(* Logix 5000 project; controller IF2_DEMO Emulate 5570 rev 20.12; software revision 20.04; part 5 of 8 *)
(* tags used below, declared in another part *)
   CIP_String_Creator : STRING;
   CIP_TimeStamp : STRING;
   CIP_TimeStamp_Day : STRING;
   CIP_TimeStamp_Month : STRING;
   CIPActive : BOOL;
   CIPAlarm_Start : BOOL;
   CIPAlarmTrigger : BOOL[32];
   CIPClarity : DINT;
   CIPFilling : BOOL[32];
   CIPTimer : TIMER[4];
   CIPValve0 : ALARM_DIGITAL;
   CIPValve1 : ALARM_DIGITAL;
   CIPValve2 : ALARM_DIGITAL;
   CIPValve3 : ALARM_DIGITAL;
   Delay : TIMER[4];
   DispenserLine : LineData;
   HMISystemClock : DINT[7];
   Menu_GOTO_dx : DINT;
   Menu_GOTO_H : DINT;
   Menu_GOTO_POS : DINT;
   MotorOverheatAlarm : ALARM_ANALOG;
   MotorTemp : DINT;
   Phase_1 : PHASE;
   Phase_2 : PHASE;
   Phase_Timer : TIMER;
   RefillLine : LineData;
   Run_Day : INT;
   Run_Hr : INT;
   Run_Min : INT;
   Run_Sec : INT;
   Run_Timer : TIMER;
   SodaCIPTanks : IPTankLevel;
   TankValue : DINT[4];
   Timer1000ms : TIMER;
   Timer100ms : TIMER;
   Timer10ms : TIMER;
   Timer1ms : TIMER;
   Timer250ms : TIMER;
   Timer500ms : TIMER;
   TimeTrigger : BOOL;
   ValveFlowOn : BOOL;
   WallClock : DINT[7];
   WC : WC[10];

PROGRAM Main   (* main routine MainRoutine *)
VAR
   Agitator : DISCRETE_2STATE := (State0Perm := 1, State1Perm := 1);
   Alarm_RapidMixStopped : ALARM_DIGITAL;
   ApplyDSTBit : DINT := 1;
   Assembly : MotionVars := (Motion := 9.0, MotionFactor := 3.0, MotionMax := 99.0);
   Blending_Discharge_Jam_Tank1 : ALARM_DIGITAL;
   Blending_Discharge_Tank1_Jam_Ack : BOOL := 1;
   Blending_Discharge_Tank1_Jam_Ind : BOOL := 1;
   Blending_Discharge_Tank1_Jam_Timer_Sim : TIMER := (PRE := 500004, ACC := 253104, EN := 1, TT := 1);
   CIP_Clarify_Sensor_Ack : BOOL;
   CIP_Clarify_Sensor_Ind : BOOL;
   CIP_Clarify_Sensor_Timer_Sim : TIMER := (PRE := 1100022, ACC := 653241, EN := 1, TT := 1);
   CIP_Clarity_Sensor : ALARM_DIGITAL;
   CIP_Drain_Valve : ALARM_DIGITAL;
   CIP_Drain_Valve_Ack : BOOL;
   CIP_Drain_Valve_Ind : BOOL;
   CIP_Drain_Valve_Timer_Sim : TIMER := (PRE := 900000, ACC := 53334, EN := 1, TT := 1);
   CIP_Supply_Motor : ALARM_ANALOG;
   CIP_Supply_Motor_Ack : BOOL;
   CIP_Supply_Motor_Ind : BOOL;
   CIP_Supply_Motor_Timer_Sim : TIMER := (PRE := 900001, ACC := 53325, EN := 1, TT := 1);
   CIP_TimeStamp_ONS : BOOL;
   CIPSteps : DINT := 5;
   Complete_Manual_Step_AUTO : TIMER := (PRE := 240000);
   Filler_Valve_3a_Ack : BOOL;
   Filler_Valve_3a_Ind : BOOL;
   Filler_Valve_3a_Timer_Sim : TIMER := (PRE := 301000, ACC := 28908, EN := 1, TT := 1);
   Filler_Valve_6B_Ack : BOOL;
   Filler_Valve_6B_Ind : BOOL;
   Filler_Valve_6B_Timer_Sim : TIMER := (PRE := 400000, ACC := 53031, EN := 1, TT := 1);
   Filling_Valve_3a : ALARM_DIGITAL;
   Filling_Valve_3a_Ack : BOOL;
   Filling_Valve_6b : ALARM_DIGITAL;
   Labeler_Motor : ALARM_ANALOG;
   Labeler_Motor_Ack : BOOL;
   Labeler_Motor_Timer_Sim : TIMER := (PRE := 200019, ACC := 51885, EN := 1, TT := 1);
   Main : MotionVars := (Motion := 30.0, MotionFactor := 1.0, MotionMax := 100.0);
   Maximum : DINT[4] := ([0] := 20000, [1] := 20000, [2] := 20000, [3] := 20000);
   Mixer_Step_6_AUTORESET : TIMER := (PRE := 15000);
   Packaging_Motor : ALARM_ANALOG;
   Packaging_Motor_Ack : BOOL;
   Packaging_Motor_Timer_Sim : TIMER := (PRE := 300222, ACC := 47541, EN := 1, TT := 1);
   Paint : MotionVars := (MotionFactor := 1.0, MotionMax := 199.0);
   repeatCIP : BOOL;
   Restart_CIP_Timer_AUTO : TIMER := (PRE := 150000, ACC := 123517, EN := 1, TT := 1);
   TempCalc : DINT[4] := ([0] := 12500, [1] := 20000, [2] := 1982, [3] := 2000);
   TempCalc2 : DINT[4] := ([0] := 20000, [1] := 20000, [2] := 7982, [3] := 8000);
   test_bit : BOOL := 1;
   Test_Pack : MotionVars := (Motion := 39.0, MotionFactor := 3.0, MotionMax := 49.0);
   Test_Toggle : BOOL;
   TestLatch : BOOL;
   trig : DINT := 20686;
   xUtility : TIMER := (PRE := 500, ACC := 313, EN := 1, TT := 1);
   xUtilityBit : DINT;
END_VAR

ROUTINE Alarms   (* ladder *)
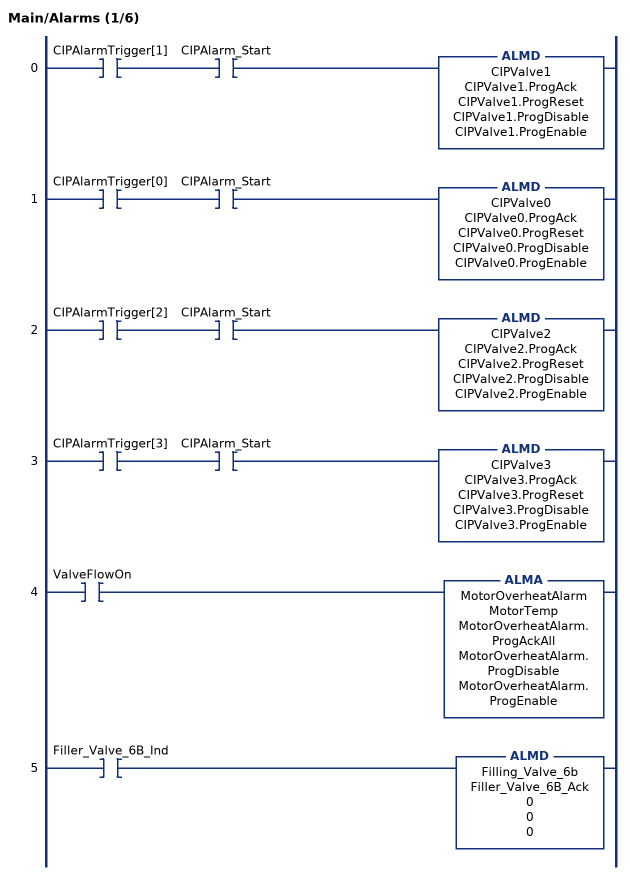
   0: XIC(CIPAlarmTrigger[1])XIC(CIPAlarm_Start)ALMD(CIPValve1,CIPValve1.ProgAck,CIPValve1.ProgReset,CIPValve1.ProgDisable,CIPValve1.ProgEnable);
   1: XIC(CIPAlarmTrigger[0])XIC(CIPAlarm_Start)ALMD(CIPValve0,CIPValve0.ProgAck,CIPValve0.ProgReset,CIPValve0.ProgDisable,CIPValve0.ProgEnable);
   2: XIC(CIPAlarmTrigger[2])XIC(CIPAlarm_Start)ALMD(CIPValve2,CIPValve2.ProgAck,CIPValve2.ProgReset,CIPValve2.ProgDisable,CIPValve2.ProgEnable);
   3: XIC(CIPAlarmTrigger[3])XIC(CIPAlarm_Start)ALMD(CIPValve3,CIPValve3.ProgAck,CIPValve3.ProgReset,CIPValve3.ProgDisable,CIPValve3.ProgEnable);
   4: XIC(ValveFlowOn)ALMA(MotorOverheatAlarm,MotorTemp,MotorOverheatAlarm.ProgAckAll,MotorOverheatAlarm.ProgDisable,MotorOverheatAlarm.ProgEnable);
   5: XIC(Filler_Valve_6B_Ind)ALMD(Filling_Valve_6b,Filler_Valve_6B_Ack,0,0,0);
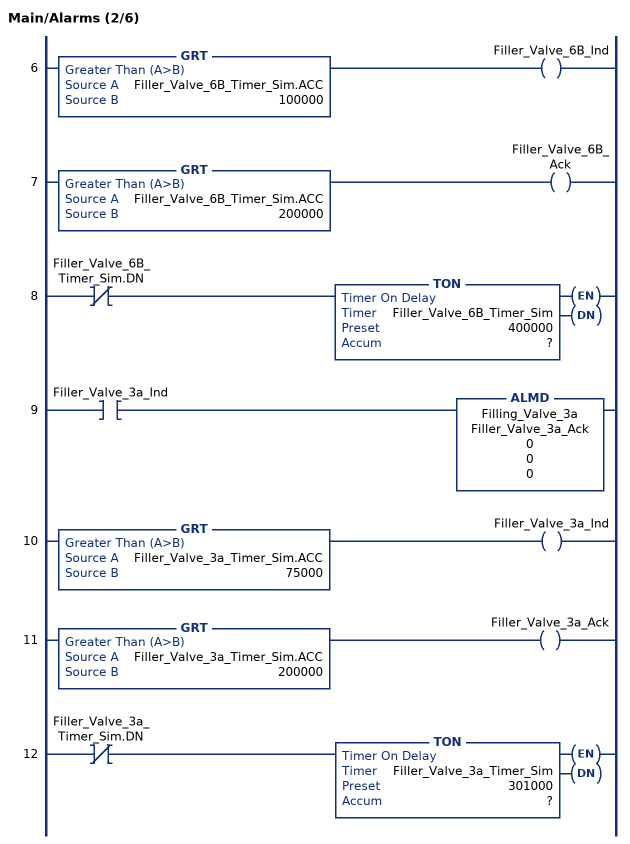
   6: GRT(Filler_Valve_6B_Timer_Sim.ACC,100000)OTE(Filler_Valve_6B_Ind);
   7: GRT(Filler_Valve_6B_Timer_Sim.ACC,200000)OTE(Filler_Valve_6B_Ack);
   8: XIO(Filler_Valve_6B_Timer_Sim.DN)TON(Filler_Valve_6B_Timer_Sim,?,?);
   9: XIC(Filler_Valve_3a_Ind)ALMD(Filling_Valve_3a,Filler_Valve_3a_Ack,0,0,0);
   10: GRT(Filler_Valve_3a_Timer_Sim.ACC,75000)OTE(Filler_Valve_3a_Ind);
   11: GRT(Filler_Valve_3a_Timer_Sim.ACC,200000)OTE(Filler_Valve_3a_Ack);
   12: XIO(Filler_Valve_3a_Timer_Sim.DN)TON(Filler_Valve_3a_Timer_Sim,?,?);
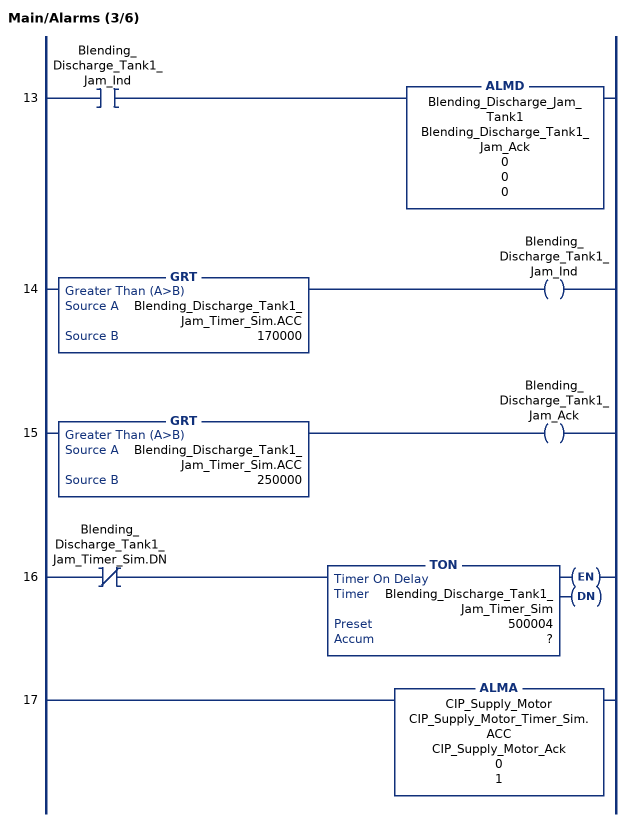
   13: XIC(Blending_Discharge_Tank1_Jam_Ind)ALMD(Blending_Discharge_Jam_Tank1,Blending_Discharge_Tank1_Jam_Ack,0,0,0);
   14: GRT(Blending_Discharge_Tank1_Jam_Timer_Sim.ACC,170000)OTE(Blending_Discharge_Tank1_Jam_Ind);
   15: GRT(Blending_Discharge_Tank1_Jam_Timer_Sim.ACC,250000)OTE(Blending_Discharge_Tank1_Jam_Ack);
   16: XIO(Blending_Discharge_Tank1_Jam_Timer_Sim.DN)TON(Blending_Discharge_Tank1_Jam_Timer_Sim,?,?);
   17: ALMA(CIP_Supply_Motor,CIP_Supply_Motor_Timer_Sim.ACC,CIP_Supply_Motor_Ack,0,1);
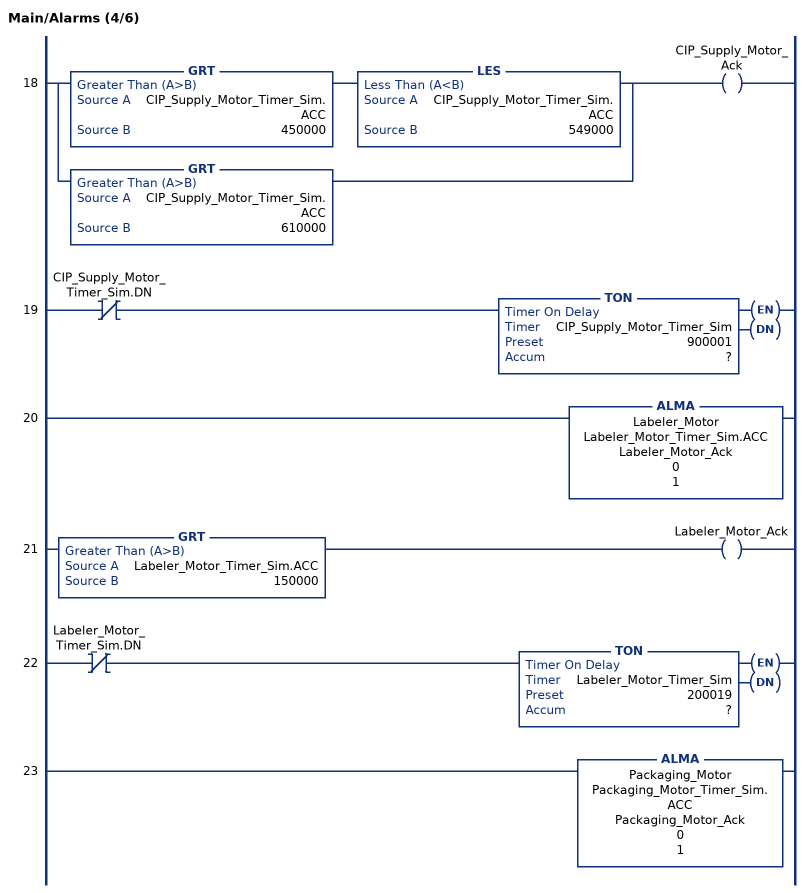
   18: [GRT(CIP_Supply_Motor_Timer_Sim.ACC,450000) LES(CIP_Supply_Motor_Timer_Sim.ACC,549000) ,GRT(CIP_Supply_Motor_Timer_Sim.ACC,610000) ]OTE(CIP_Supply_Motor_Ack);
   19: XIO(CIP_Supply_Motor_Timer_Sim.DN)TON(CIP_Supply_Motor_Timer_Sim,?,?);
   20: ALMA(Labeler_Motor,Labeler_Motor_Timer_Sim.ACC,Labeler_Motor_Ack,0,1);
   21: GRT(Labeler_Motor_Timer_Sim.ACC,150000)OTE(Labeler_Motor_Ack);
   22: XIO(Labeler_Motor_Timer_Sim.DN)TON(Labeler_Motor_Timer_Sim,?,?);
   23: ALMA(Packaging_Motor,Packaging_Motor_Timer_Sim.ACC,Packaging_Motor_Ack,0,1);
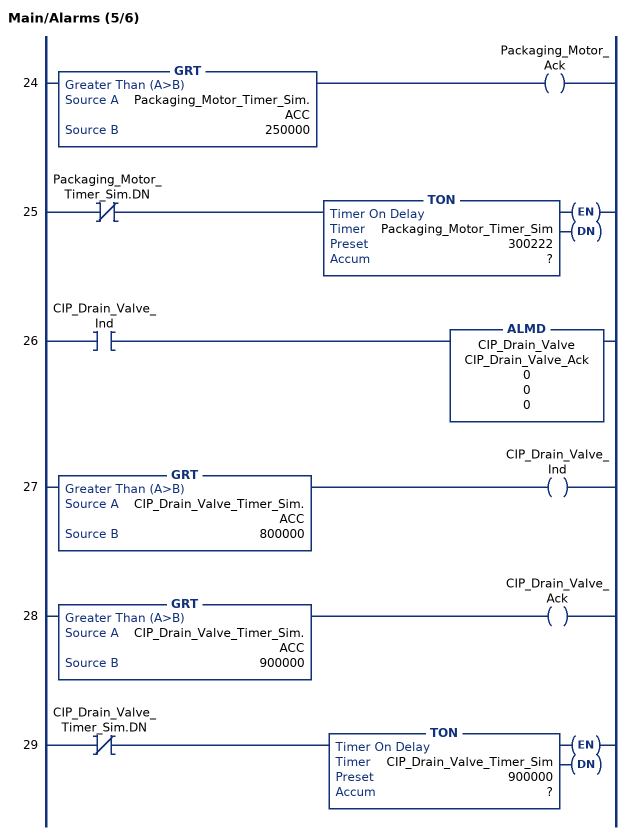
   24: GRT(Packaging_Motor_Timer_Sim.ACC,250000)OTE(Packaging_Motor_Ack);
   25: XIO(Packaging_Motor_Timer_Sim.DN)TON(Packaging_Motor_Timer_Sim,?,?);
   26: XIC(CIP_Drain_Valve_Ind)ALMD(CIP_Drain_Valve,CIP_Drain_Valve_Ack,0,0,0);
   27: GRT(CIP_Drain_Valve_Timer_Sim.ACC,800000)OTE(CIP_Drain_Valve_Ind);
   28: GRT(CIP_Drain_Valve_Timer_Sim.ACC,900000)OTE(CIP_Drain_Valve_Ack);
   29: XIO(CIP_Drain_Valve_Timer_Sim.DN)TON(CIP_Drain_Valve_Timer_Sim,?,?);
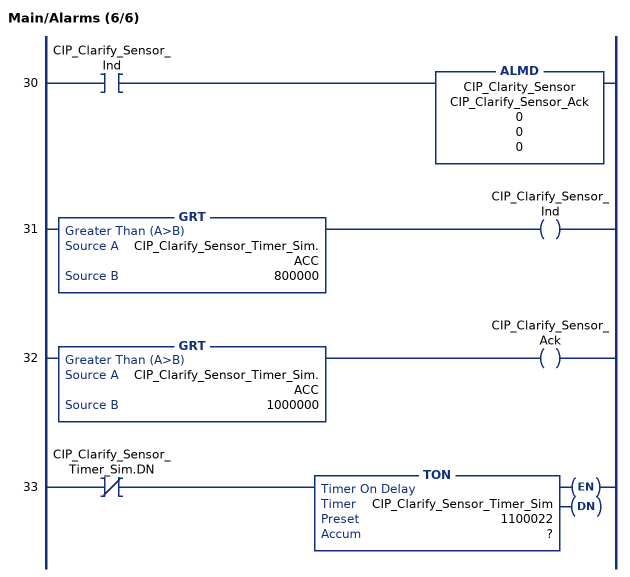
   30: XIC(CIP_Clarify_Sensor_Ind)ALMD(CIP_Clarity_Sensor,CIP_Clarify_Sensor_Ack,0,0,0);
   31: GRT(CIP_Clarify_Sensor_Timer_Sim.ACC,800000)OTE(CIP_Clarify_Sensor_Ind);
   32: GRT(CIP_Clarify_Sensor_Timer_Sim.ACC,1000000)OTE(CIP_Clarify_Sensor_Ack);
   33: XIO(CIP_Clarify_Sensor_Timer_Sim.DN)TON(CIP_Clarify_Sensor_Timer_Sim,?,?);
END_ROUTINE

ROUTINE CIP   (* ladder *)
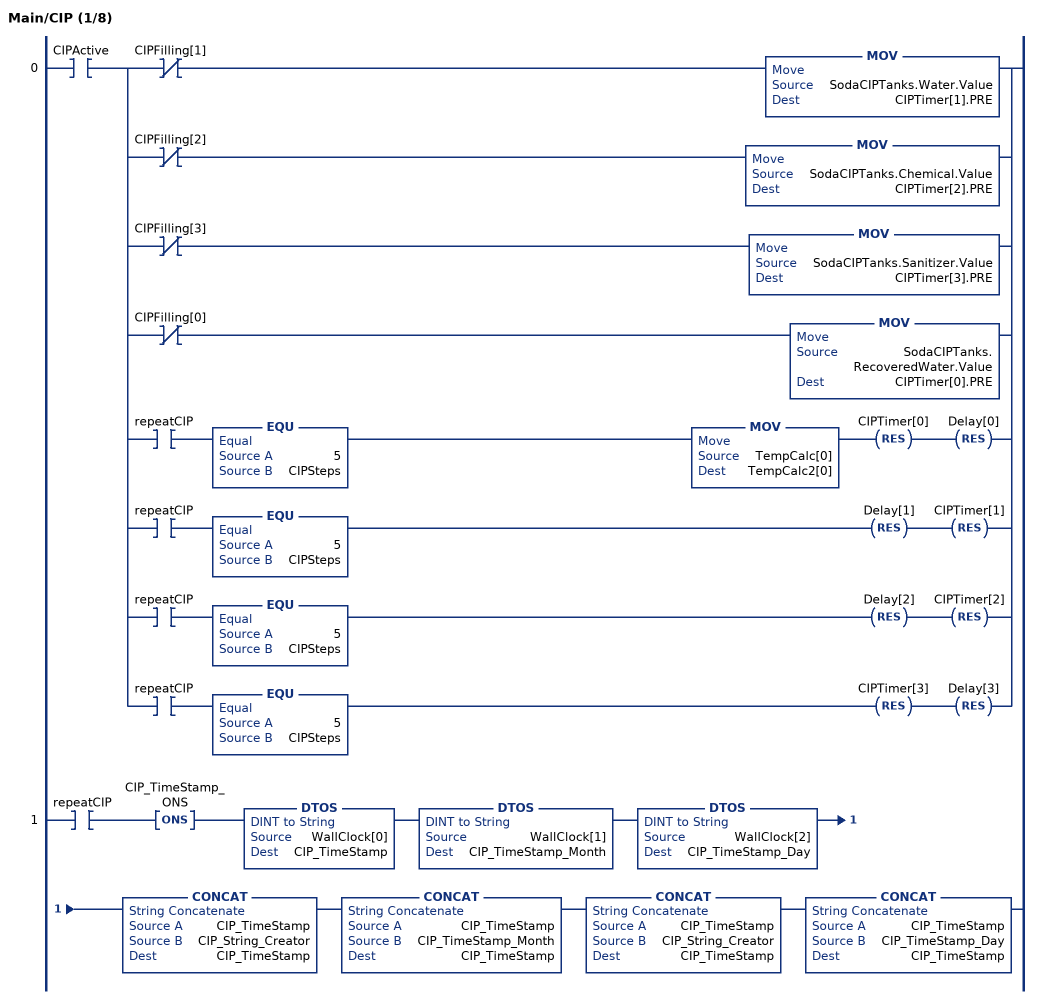
   0: XIC(CIPActive)[XIO(CIPFilling[1]) MOV(SodaCIPTanks.Water.Value,CIPTimer[1].PRE) ,[XIO(CIPFilling[2]) MOV(SodaCIPTanks.Chemical.Value,CIPTimer[2].PRE) ,XIO(CIPFilling[3]) MOV(SodaCIPTanks.Sanitizer.Value,CIPTimer[3].PRE) ,XIO(CIPFilling[0]) MOV(SodaCIPTanks.RecoveredWater.Value,CIPTimer[0].PRE) ,XIC(repeatCIP) EQU(5,CIPSteps) MOV(TempCalc[0],TempCalc2[0]) RES(CIPTimer[0]) RES(Delay[0]) ,XIC(repeatCIP) EQU(5,CIPSteps) RES(Delay[1]) RES(CIPTimer[1]) ,XIC(repeatCIP) EQU(5,CIPSteps) RES(Delay[2]) RES(CIPTimer[2]) ,XIC(repeatCIP) EQU(5,CIPSteps) RES(CIPTimer[3]) RES(Delay[3]) ] ];
   1: XIC(repeatCIP)ONS(CIP_TimeStamp_ONS)DTOS(WallClock[0],CIP_TimeStamp)DTOS(WallClock[1],CIP_TimeStamp_Month)DTOS(WallClock[2],CIP_TimeStamp_Day)CONCAT(CIP_TimeStamp,CIP_String_Creator,CIP_TimeStamp)CONCAT(CIP_TimeStamp,CIP_TimeStamp_Month,CIP_TimeStamp)CONCAT(CIP_TimeStamp,CIP_String_Creator,CIP_TimeStamp)CONCAT(CIP_TimeStamp,CIP_TimeStamp_Day,CIP_TimeStamp);
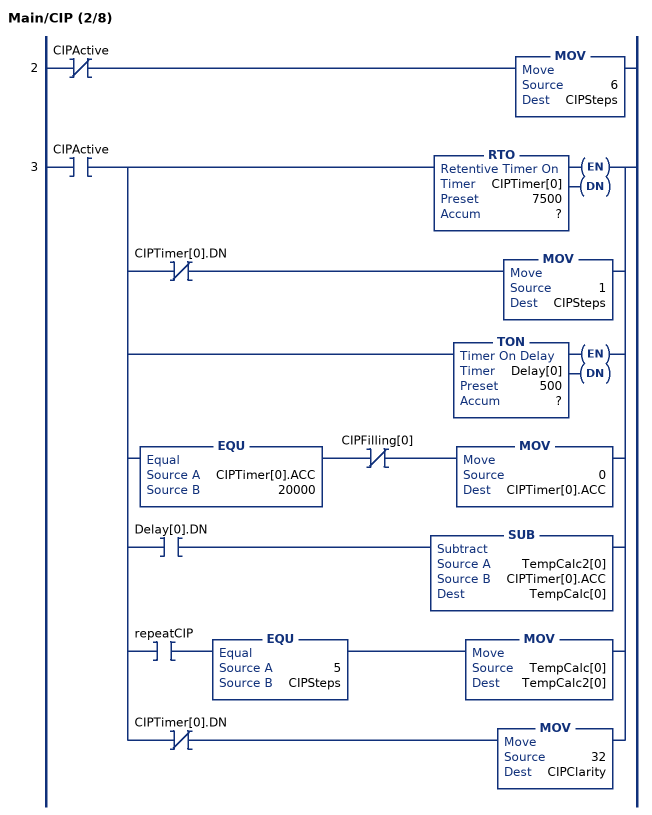
   2: XIO(CIPActive)MOV(6,CIPSteps);
   3: XIC(CIPActive)[RTO(CIPTimer[0],?,?) ,XIO(CIPTimer[0].DN) MOV(1,CIPSteps) ,TON(Delay[0],?,?) ,EQU(CIPTimer[0].ACC,20000) XIO(CIPFilling[0]) MOV(0,CIPTimer[0].ACC) ,XIC(Delay[0].DN) SUB(TempCalc2[0],CIPTimer[0].ACC,TempCalc[0]) ,XIC(repeatCIP) EQU(5,CIPSteps) MOV(TempCalc[0],TempCalc2[0]) ,XIO(CIPTimer[0].DN) MOV(32,CIPClarity) ];
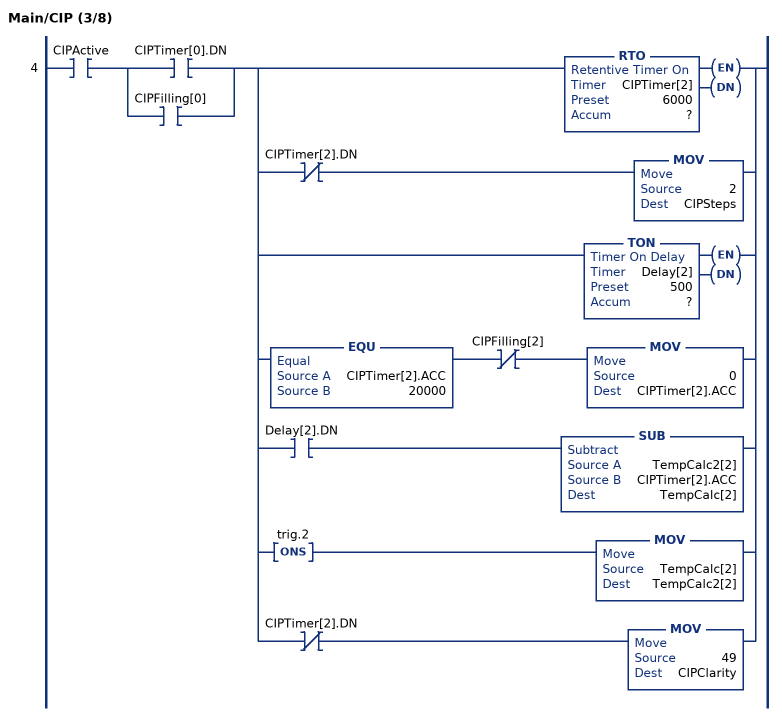
   4: XIC(CIPActive)[XIC(CIPTimer[0].DN) ,XIC(CIPFilling[0]) ][RTO(CIPTimer[2],?,?) ,XIO(CIPTimer[2].DN) MOV(2,CIPSteps) ,TON(Delay[2],?,?) ,EQU(CIPTimer[2].ACC,20000) XIO(CIPFilling[2]) MOV(0,CIPTimer[2].ACC) ,XIC(Delay[2].DN) SUB(TempCalc2[2],CIPTimer[2].ACC,TempCalc[2]) ,ONS(trig.2) MOV(TempCalc[2],TempCalc2[2]) ,XIO(CIPTimer[2].DN) MOV(49,CIPClarity) ];
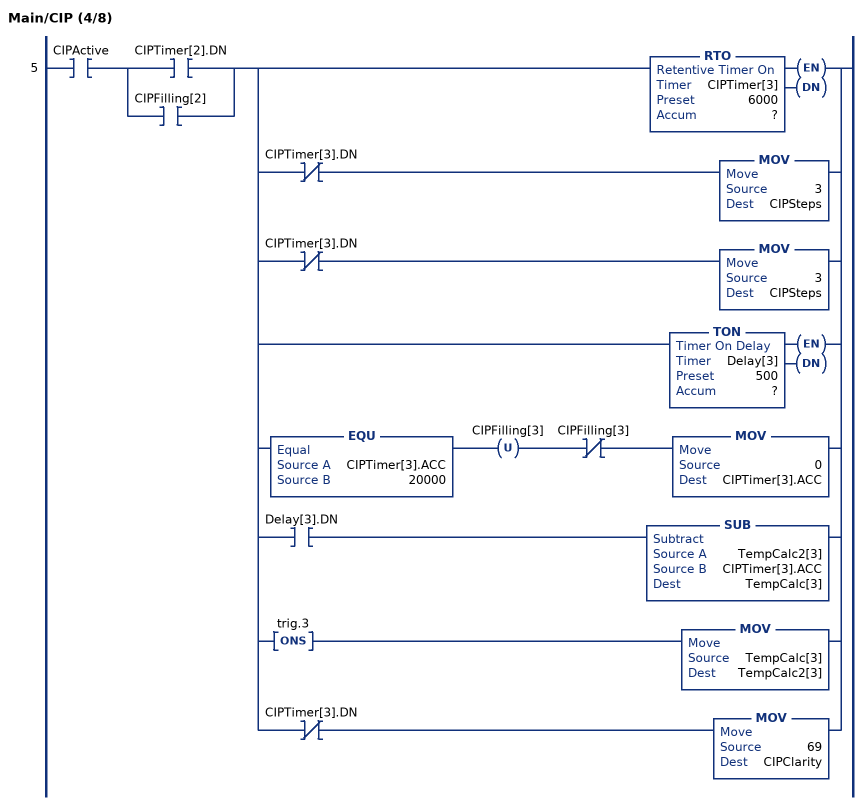
   5: XIC(CIPActive)[XIC(CIPTimer[2].DN) ,XIC(CIPFilling[2]) ][RTO(CIPTimer[3],?,?) ,XIO(CIPTimer[3].DN) MOV(3,CIPSteps) ,XIO(CIPTimer[3].DN) MOV(3,CIPSteps) ,TON(Delay[3],?,?) ,EQU(CIPTimer[3].ACC,20000) OTU(CIPFilling[3]) XIO(CIPFilling[3]) MOV(0,CIPTimer[3].ACC) ,XIC(Delay[3].DN) SUB(TempCalc2[3],CIPTimer[3].ACC,TempCalc[3]) ,ONS(trig.3) MOV(TempCalc[3],TempCalc2[3]) ,XIO(CIPTimer[3].DN) MOV(69,CIPClarity) ];
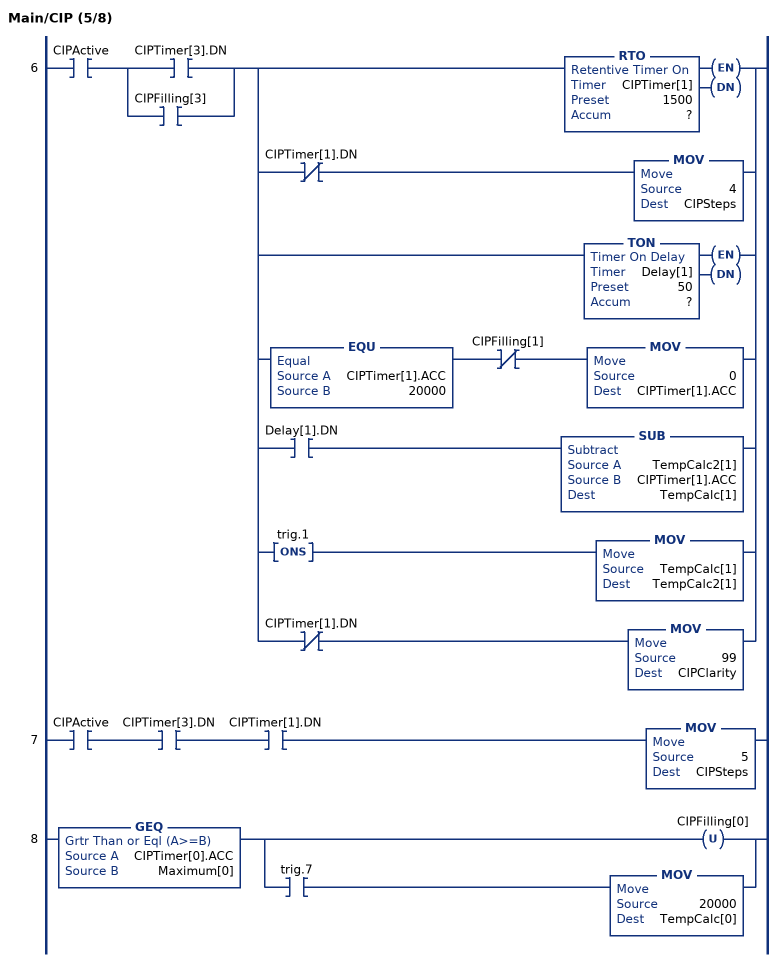
   6: XIC(CIPActive)[XIC(CIPTimer[3].DN) ,XIC(CIPFilling[3]) ][RTO(CIPTimer[1],?,?) ,XIO(CIPTimer[1].DN) MOV(4,CIPSteps) ,TON(Delay[1],?,?) ,EQU(CIPTimer[1].ACC,20000) XIO(CIPFilling[1]) MOV(0,CIPTimer[1].ACC) ,XIC(Delay[1].DN) SUB(TempCalc2[1],CIPTimer[1].ACC,TempCalc[1]) ,ONS(trig.1) MOV(TempCalc[1],TempCalc2[1]) ,XIO(CIPTimer[1].DN) MOV(99,CIPClarity) ];
   7: XIC(CIPActive)XIC(CIPTimer[3].DN)XIC(CIPTimer[1].DN)MOV(5,CIPSteps);
   8: GEQ(CIPTimer[0].ACC,Maximum[0])[OTU(CIPFilling[0]) ,XIC(trig.7) MOV(20000,TempCalc[0]) ];
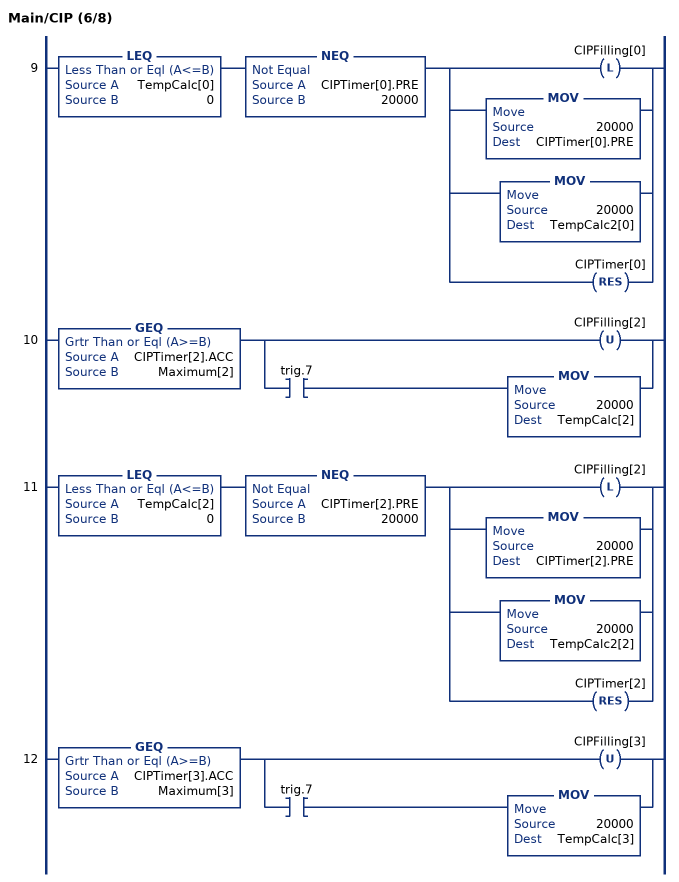
   9: LEQ(TempCalc[0],0)NEQ(CIPTimer[0].PRE,20000)[OTL(CIPFilling[0]) ,MOV(20000,CIPTimer[0].PRE) ,MOV(20000,TempCalc2[0]) ,RES(CIPTimer[0]) ];
   10: GEQ(CIPTimer[2].ACC,Maximum[2])[OTU(CIPFilling[2]) ,XIC(trig.7) MOV(20000,TempCalc[2]) ];
   11: LEQ(TempCalc[2],0)NEQ(CIPTimer[2].PRE,20000)[OTL(CIPFilling[2]) ,MOV(20000,CIPTimer[2].PRE) ,MOV(20000,TempCalc2[2]) ,RES(CIPTimer[2]) ];
   12: GEQ(CIPTimer[3].ACC,Maximum[3])[OTU(CIPFilling[3]) ,XIC(trig.7) MOV(20000,TempCalc[3]) ];
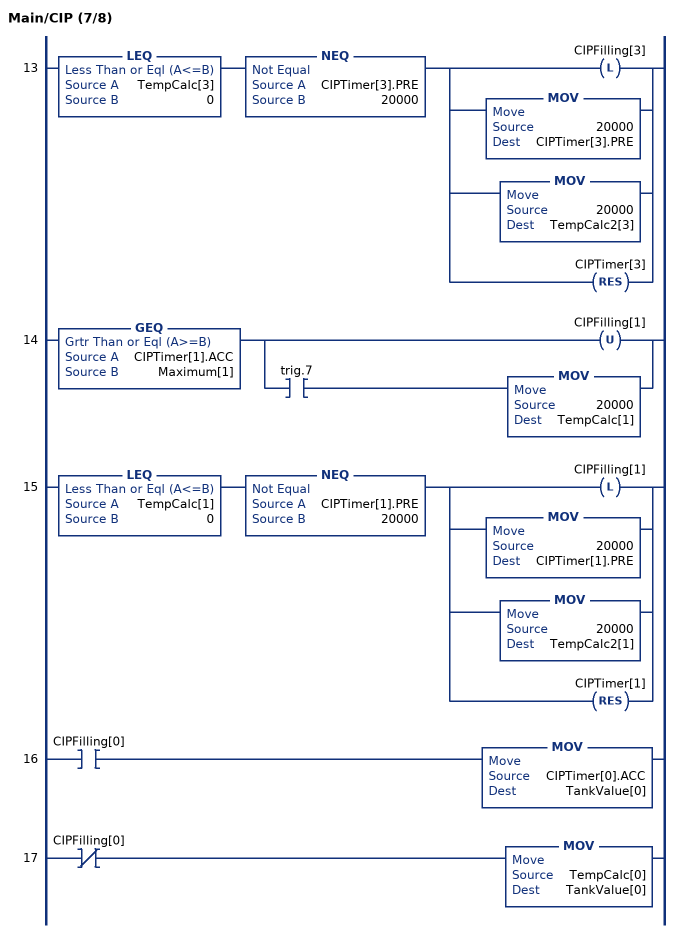
   13: LEQ(TempCalc[3],0)NEQ(CIPTimer[3].PRE,20000)[OTL(CIPFilling[3]) ,MOV(20000,CIPTimer[3].PRE) ,MOV(20000,TempCalc2[3]) ,RES(CIPTimer[3]) ];
   14: GEQ(CIPTimer[1].ACC,Maximum[1])[OTU(CIPFilling[1]) ,XIC(trig.7) MOV(20000,TempCalc[1]) ];
   15: LEQ(TempCalc[1],0)NEQ(CIPTimer[1].PRE,20000)[OTL(CIPFilling[1]) ,MOV(20000,CIPTimer[1].PRE) ,MOV(20000,TempCalc2[1]) ,RES(CIPTimer[1]) ];
   16: XIC(CIPFilling[0])MOV(CIPTimer[0].ACC,TankValue[0]);
   17: XIO(CIPFilling[0])MOV(TempCalc[0],TankValue[0]);
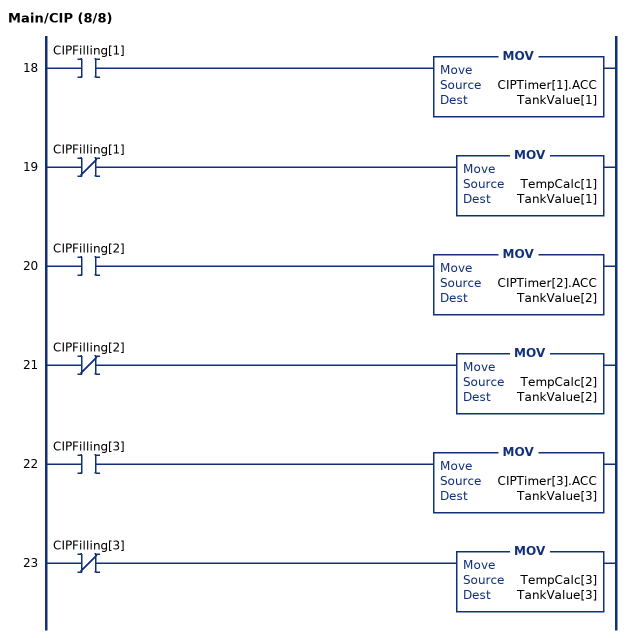
   18: XIC(CIPFilling[1])MOV(CIPTimer[1].ACC,TankValue[1]);
   19: XIO(CIPFilling[1])MOV(TempCalc[1],TankValue[1]);
   20: XIC(CIPFilling[2])MOV(CIPTimer[2].ACC,TankValue[2]);
   21: XIO(CIPFilling[2])MOV(TempCalc[2],TankValue[2]);
   22: XIC(CIPFilling[3])MOV(CIPTimer[3].ACC,TankValue[3]);
   23: XIO(CIPFilling[3])MOV(TempCalc[3],TankValue[3]);
END_ROUTINE

ROUTINE MainRoutine   (* ladder *)
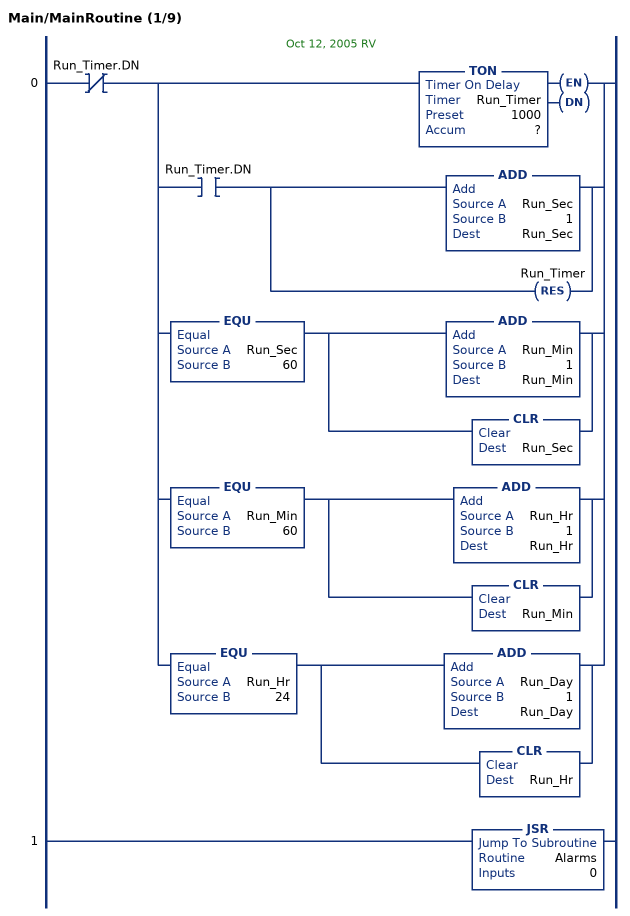
   // Oct 12, 2005 RV
   0: XIO(Run_Timer.DN)[TON(Run_Timer,?,?) ,XIC(Run_Timer.DN) [ADD(Run_Sec,1,Run_Sec) ,RES(Run_Timer) ] ,EQU(Run_Sec,60) [ADD(Run_Min,1,Run_Min) ,CLR(Run_Sec) ] ,EQU(Run_Min,60) [ADD(Run_Hr,1,Run_Hr) ,CLR(Run_Min) ] ,EQU(Run_Hr,24) [ADD(Run_Day,1,Run_Day) ,CLR(Run_Hr) ] ];
   1: JSR(Alarms,0);
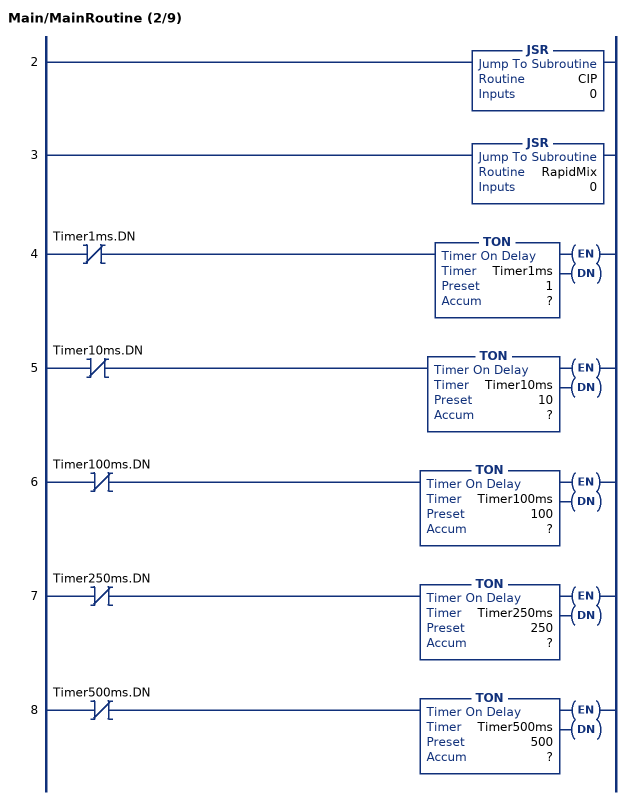
   2: JSR(CIP,0);
   3: JSR(RapidMix,0);
   4: XIO(Timer1ms.DN)TON(Timer1ms,?,?);
   5: XIO(Timer10ms.DN)TON(Timer10ms,?,?);
   6: XIO(Timer100ms.DN)TON(Timer100ms,?,?);
   7: XIO(Timer250ms.DN)TON(Timer250ms,?,?);
   8: XIO(Timer500ms.DN)TON(Timer500ms,?,?);
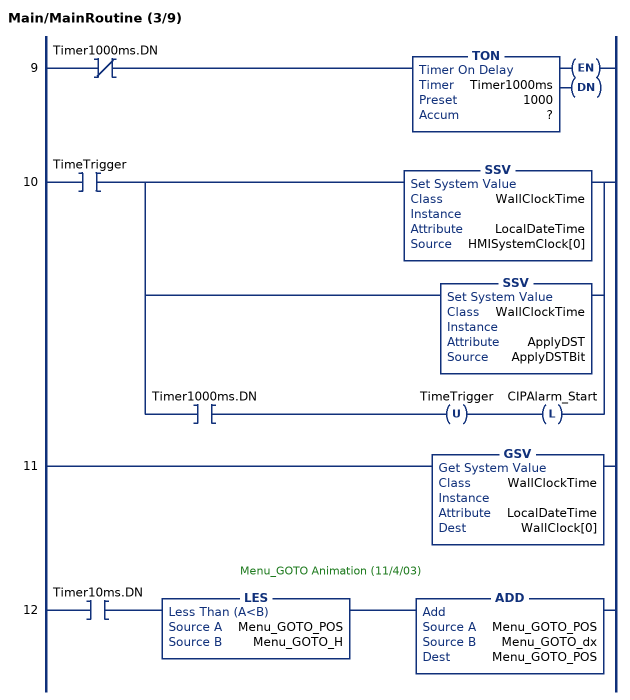
   9: XIO(Timer1000ms.DN)TON(Timer1000ms,?,?);
   10: XIC(TimeTrigger)[SSV(WallClockTime,,LocalDateTime,HMISystemClock[0]) ,SSV(WallClockTime,,ApplyDST,ApplyDSTBit) ,XIC(Timer1000ms.DN) OTU(TimeTrigger) OTL(CIPAlarm_Start) ];
   11: GSV(WallClockTime,,LocalDateTime,WallClock[0]);
   // Menu_GOTO Animation (11/4/03)
   12: XIC(Timer10ms.DN)LES(Menu_GOTO_POS,Menu_GOTO_H)ADD(Menu_GOTO_POS,Menu_GOTO_dx,Menu_GOTO_POS);
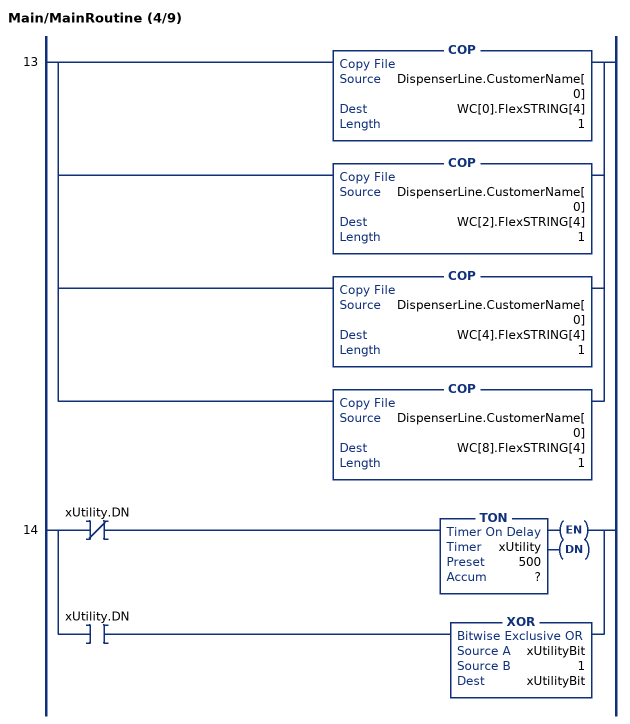
   13: [COP(DispenserLine.CustomerName[0],WC[0].FlexSTRING[4],1) ,COP(DispenserLine.CustomerName[0],WC[2].FlexSTRING[4],1) ,COP(DispenserLine.CustomerName[0],WC[4].FlexSTRING[4],1) ,COP(DispenserLine.CustomerName[0],WC[8].FlexSTRING[4],1) ];
   14: [XIO(xUtility.DN) TON(xUtility,?,?) ,XIC(xUtility.DN) XOR(xUtilityBit,1,xUtilityBit) ];
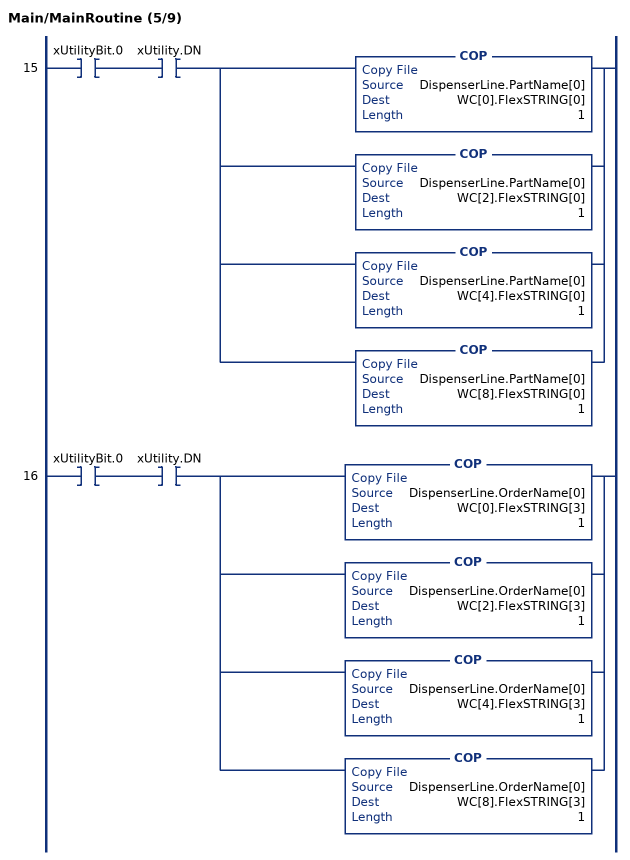
   15: XIC(xUtilityBit.0)XIC(xUtility.DN)[COP(DispenserLine.PartName[0],WC[0].FlexSTRING[0],1) ,COP(DispenserLine.PartName[0],WC[2].FlexSTRING[0],1) ,COP(DispenserLine.PartName[0],WC[4].FlexSTRING[0],1) ,COP(DispenserLine.PartName[0],WC[8].FlexSTRING[0],1) ];
   16: XIC(xUtilityBit.0)XIC(xUtility.DN)[COP(DispenserLine.OrderName[0],WC[0].FlexSTRING[3],1) ,COP(DispenserLine.OrderName[0],WC[2].FlexSTRING[3],1) ,COP(DispenserLine.OrderName[0],WC[4].FlexSTRING[3],1) ,COP(DispenserLine.OrderName[0],WC[8].FlexSTRING[3],1) ];
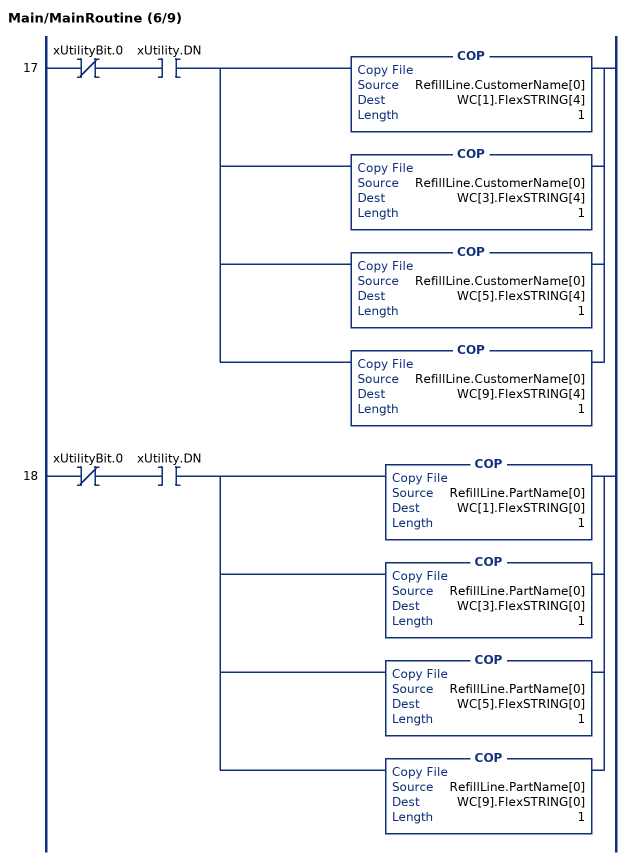
   17: XIO(xUtilityBit.0)XIC(xUtility.DN)[COP(RefillLine.CustomerName[0],WC[1].FlexSTRING[4],1) ,COP(RefillLine.CustomerName[0],WC[3].FlexSTRING[4],1) ,COP(RefillLine.CustomerName[0],WC[5].FlexSTRING[4],1) ,COP(RefillLine.CustomerName[0],WC[9].FlexSTRING[4],1) ];
   18: XIO(xUtilityBit.0)XIC(xUtility.DN)[COP(RefillLine.PartName[0],WC[1].FlexSTRING[0],1) ,COP(RefillLine.PartName[0],WC[3].FlexSTRING[0],1) ,COP(RefillLine.PartName[0],WC[5].FlexSTRING[0],1) ,COP(RefillLine.PartName[0],WC[9].FlexSTRING[0],1) ];
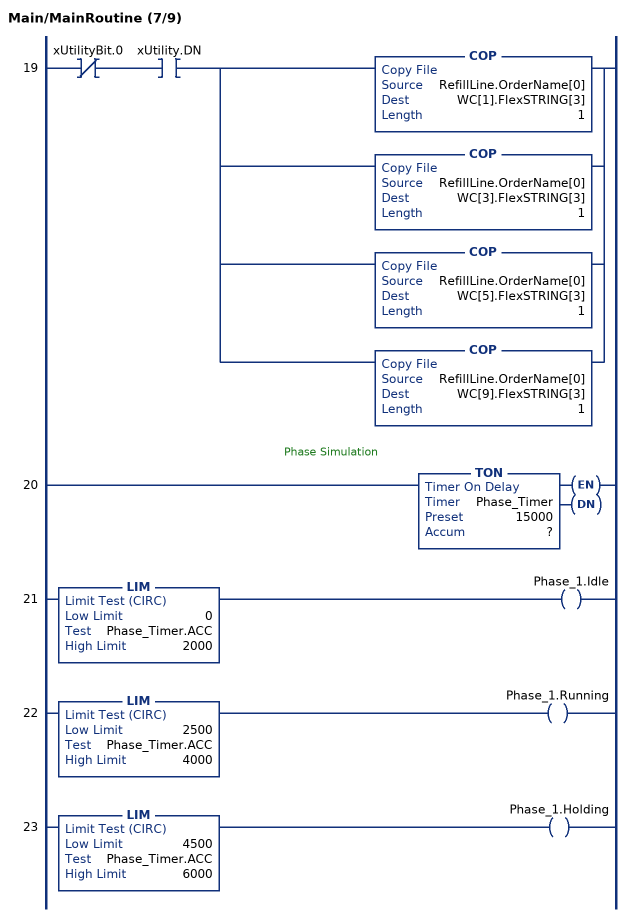
   19: XIO(xUtilityBit.0)XIC(xUtility.DN)[COP(RefillLine.OrderName[0],WC[1].FlexSTRING[3],1) ,COP(RefillLine.OrderName[0],WC[3].FlexSTRING[3],1) ,COP(RefillLine.OrderName[0],WC[5].FlexSTRING[3],1) ,COP(RefillLine.OrderName[0],WC[9].FlexSTRING[3],1) ];
   // Phase Simulation
   20: TON(Phase_Timer,?,?);
   21: LIM(0,Phase_Timer.ACC,2000)OTE(Phase_1.Idle);
   22: LIM(2500,Phase_Timer.ACC,4000)OTE(Phase_1.Running);
   23: LIM(4500,Phase_Timer.ACC,6000)OTE(Phase_1.Holding);
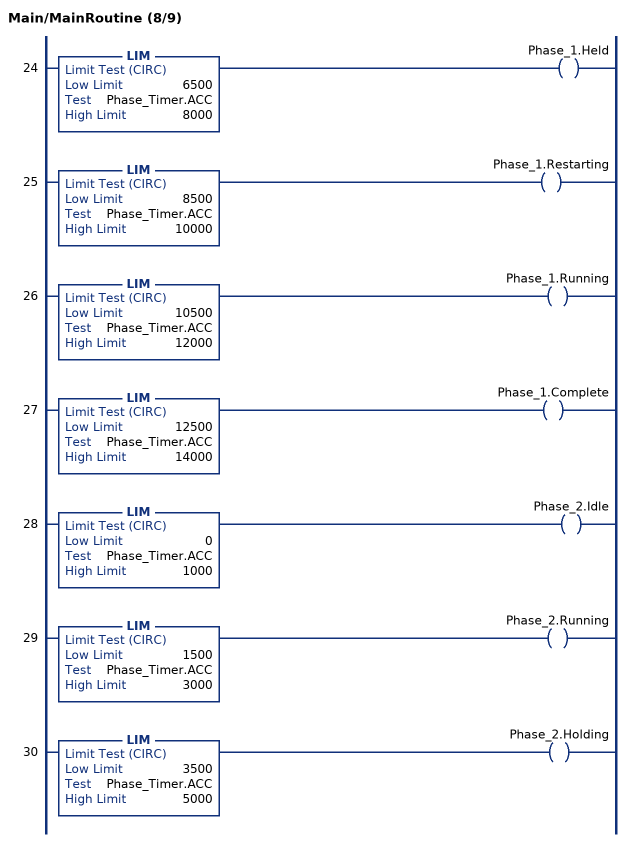
   24: LIM(6500,Phase_Timer.ACC,8000)OTE(Phase_1.Held);
   25: LIM(8500,Phase_Timer.ACC,10000)OTE(Phase_1.Restarting);
   26: LIM(10500,Phase_Timer.ACC,12000)OTE(Phase_1.Running);
   27: LIM(12500,Phase_Timer.ACC,14000)OTE(Phase_1.Complete);
   28: LIM(0,Phase_Timer.ACC,1000)OTE(Phase_2.Idle);
   29: LIM(1500,Phase_Timer.ACC,3000)OTE(Phase_2.Running);
   30: LIM(3500,Phase_Timer.ACC,5000)OTE(Phase_2.Holding);
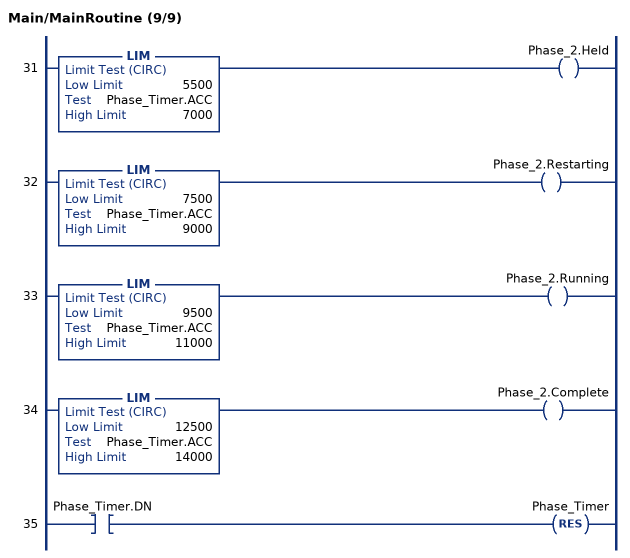
   31: LIM(5500,Phase_Timer.ACC,7000)OTE(Phase_2.Held);
   32: LIM(7500,Phase_Timer.ACC,9000)OTE(Phase_2.Restarting);
   33: LIM(9500,Phase_Timer.ACC,11000)OTE(Phase_2.Running);
   34: LIM(12500,Phase_Timer.ACC,14000)OTE(Phase_2.Complete);
   35: XIC(Phase_Timer.DN)RES(Phase_Timer);
END_ROUTINE
